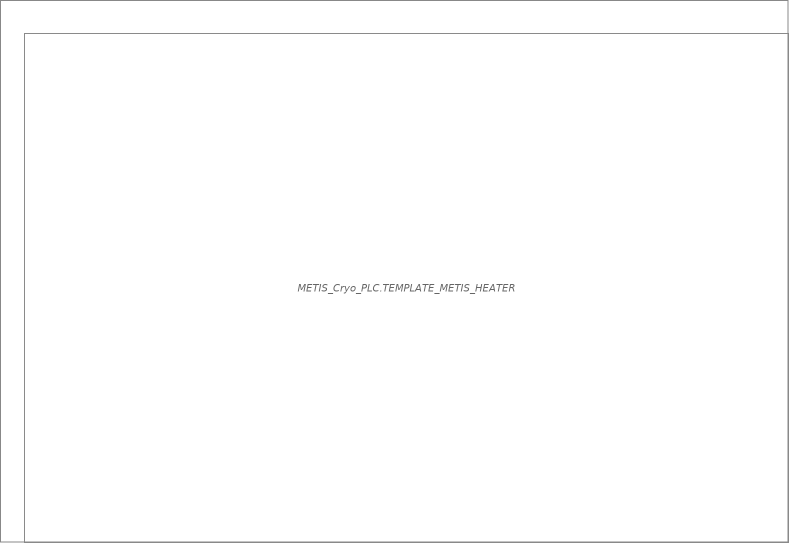
VISUALIZATION VISU_Detector_Heater  // 789x543
    Frame (24,33 765x510)
        shows METIS_Cryo_PLC.TEMPLATE_METIS_HEATER(m_instance := MAIN.nott_cryo_ctrl.nott_heaters.h_detector)
END_VISUALIZATION

(* stored: Version 1.1.0.1, ProductVersion 3.1.4026.18
   Visu VISU_Detector_Heater: Id {7a2387f8-b358-4045-9624-eb300af7d08a} *)
